FUNCTION_BLOCK ABSTRACT Device EXTENDS Core.Object IMPLEMENTS IDevice
VAR
	_Parent : ISimulatable;
	
	_LocalSimulationMode : BOOL;
END_VAR

METHOD EmergncyStop
END_METHOD

METHOD FB_init : BOOL
VAR_INPUT
	(* if TRUE, the retain variables are initialized (warm start / cold start)*)
	bInitRetains	: BOOL;
	(* if TRUE, the instance afterwards gets moved into the copy code (online change)*)
	bInCopyCode	: BOOL;
	parent : ISimulatable;
END_VAR
VAR
	parentNullException : Core.ArgumentNullException;
END_VAR
IF parent = 0 THEN
	parentNullException.Throw(CurrentNamespace.Name, ClassName, __POUNAME(), __POSITION(), 'parent');
END_IF

_Parent := parent;
END_METHOD

METHOD HandleFault
END_METHOD

METHOD Initialize : BOOL
Initialize := TRUE;
END_METHOD

{attribute 'monitoring' := 'call'}
{attribute 'OPC.UA.DA' := '1'}
{attribute 'OPC.UA.DA.Access' := '1'}
PROPERTY FINAL LocalSimulationMode : BOOL
GET
LocalSimulationMode := _LocalSimulationMode;
END_GET
END_PROPERTY

{attribute 'monitoring' := 'call'}
{attribute 'OPC.UA.DA' := '1'}
{attribute 'OPC.UA.DA.Access' := '1'}
PROPERTY FINAL SimulationMode : BOOL
GET
SimulationMode := LocalSimulationMode OR_ELSE _Parent.SimulationMode;
END_GET
END_PROPERTY

END_FUNCTION_BLOCK

(* stored: Version 1.1.0.1
   POU Device: Id {6944c97a-6dfb-4e2d-8c23-cd64be3e6040}, SpecialFunc None
   Method EmergncyStop: Id {22ca83d7-704d-4f77-89d2-d4e616bf8560}
   Method FB_init: Id {36bb165b-809d-4593-8113-eb7a691f3742}
   Method HandleFault: Id {906e7f98-c375-4200-9ed6-8d8d64b44f14}
   Method Initialize: Id {edfb1f93-c3bf-4edc-ac25-e58b01738aba}
   Property LocalSimulationMode: Id {bb136f24-8aac-4730-a3e6-c2af4208b900}
   Get Get: Id {b83861ee-0ebc-46e7-a856-c922a39df953}
   Property SimulationMode: Id {1349ab81-4e65-4f59-87e9-1d9b173f728c}
   Get Get: Id {fbddca9d-8f56-4f1a-8c81-6f78d14aee8c} *)
